FUNCTION_BLOCK FB_SIM_RS_COMM_DUMMY EXTENDS FB_SIM_RS_COMM_BASE
VAR_INPUT
END_VAR
VAR_OUTPUT
END_VAR
VAR
	//
	// TODO: Status structure for <devices>.
	// See also: FB_SIM_RS_COMM_LAKESHORE.
	//
	
	fbTimer:		TON;	// Used for ramps etc.

END_VAR

M_ActivityDo();	// Implement ramps, etc, if any

METHOD M_ActivityDo
VAR_INPUT
END_VAR
// TODO User: Implement ramps, if any.
END_METHOD

METHOD M_GetSimReply : STRING(255)
VAR_INPUT
	{attribute 'OPC.UA.DA' := '0'}
	in_sReceived:	STRING(255);		// String received from a client
END_VAR
VAR
	sReply:	STRING(255);
	lrVal:	LREAL;
	i:		INT;
    fbFormat   : FB_FormatString;
    sOut       : T_MaxString;
	nCh:	INT := 8;	// Number of channels for models 218 and 224
END_VAR
// TODO User: Implement simulated replies.

// Dummy empty reply
M_GetSimReply	:= in_sReplySuffix;
END_METHOD

END_FUNCTION_BLOCK

(* stored: Version 1.1.0.1, ProductVersion 3.1.4024.3
   POU FB_SIM_RS_COMM_DUMMY: Id {78ec6e3a-ce3c-4295-b8dc-c355f2704bf3}, SpecialFunc None
   Method M_ActivityDo: Id {7f03c4d6-d27a-4edc-a39c-4fcf4fce9948}
   Method M_GetSimReply: Id {558b92bd-7e8f-440e-bfa8-d37b7ddaa29f} *)
